{attribute 'GeneratedUsingTerminal: EPP7342-0002-0016'}
{attribute addProperty BoxType "EPP7342-0002-0016"}
{attribute addProperty Id "EnableBOOL1ResetBOOL1Reduce_torqueBOOL1"}
{attribute addProperty CRC "3376996594"}
{attribute addProperty Size "3"}
TYPE Control_C948E0F2 :
STRUCT
	{attribute addProperty Name "Enable"}
	Enable : BOOL;
	{attribute addProperty Name "Reset"}
	Reset : BOOL;
	{attribute addProperty Name "Reduce_torque"}
	Reduce_torque : BOOL;
END_STRUCT
END_TYPE

(* stored: Version 1.2.0.0, ProductVersion 3.1.4024.9
   DUT Control_C948E0F2: Id {2b5477af-fdae-474a-b03a-3a3c7c0e830d} *)
